// TwinCAT 3 PLC project PLC
// ProgramVersion: 3.1.4024.0
// libraries:
//   Tc2_Standard, * (Beckhoff Automation GmbH)
//   Tc2_System, * (Beckhoff Automation GmbH)
//   Tc3_Module, * (Beckhoff Automation GmbH)
// project tree:
//   / PlcTask1.TcTTO, PlcTask2.TcTTO
//   POUs/ MAIN_ST.TcPOU, MAIN_CFC.TcPOU, ProductionAnalytics.TcPOU
// real-time tasks:
//   TASK PlcTask1: cycle T#10ms, priority 20, ADS port 350
//   TASK PlcTask2: cycle T#10ms, priority 1, ADS port 351

CONFIGURATION PLC
    RESOURCE PLC ON TwinCAT3
        TASK PlcTask1(INTERVAL := T#10ms, PRIORITY := 20);
        TASK PlcTask2(INTERVAL := T#10ms, PRIORITY := 1);
        PROGRAM MAIN_ST WITH PlcTask1 : MAIN_ST;
        PROGRAM MAIN_CFC WITH PlcTask2 : MAIN_CFC;
    END_RESOURCE
END_CONFIGURATION

// ---- POUs/MAIN_ST.TcPOU
PROGRAM MAIN_ST
VAR
	ProductionAnalytics		:	ProductionAnalytics;
	UnsortArray		: ARRAY[1..10] OF REAL := [5, 3, 8, 5, 6, 5, 5, 23, 5, 9];
	SortedArray		: ARRAY[1..10] OF REAL;
	
	Sort			: BOOL;
	GetMean			: BOOL;
	GetStdDev		: BOOL;
	GetTotal		: BOOL;
	GetMax			: BOOL;
	GetMin			: BOOL;
	FindItem		: BOOL;
	Mean			: REAL;
	StdDev			: REAL;
	Total			: REAL;
	MaxItem			: REAL;
	MinItem			: REAL;
	FoundItemIdx	: UINT;
	ItemFound		: BOOL;
	ValidInput		: BOOL;
	IsSorted		: BOOL;
END_VAR

ProductionAnalytics(DataArray:=UnsortArray);
IF GetMean THEN
	Mean := ProductionAnalytics.GetMean();
ELSIF GetStdDev THEN
	StdDev := ProductionAnalytics.GetStdDev();
ELSIF GetTotal THEN
	Total := ProductionAnalytics.GetTotal();
ELSIF FindItem THEN
	ProductionAnalytics.FindItem( SearchValue := 23, StartIndex := 1, Endindex := 10,
								  FoundIndex => FoundItemIdx , 
								  Found => ItemFound, 
								  ValidInput => ValidInput);
ELSIF Sort THEN
	ProductionAnalytics.Sort(SortedArray => SortedArray, 
							 IsSorted => IsSorted, 
							 ValidInput => ValidInput);
ELSIF GetMax THEN
	MaxItem := ProductionAnalytics.GetMaxItem();

ELSIF GetMin THEN
	MinItem := ProductionAnalytics.GetMinItem();
END_IF

END_PROGRAM

// ---- POUs/ProductionAnalytics.TcPOU
FUNCTION_BLOCK ProductionAnalytics

VAR_IN_OUT
	DataArray 		: ARRAY[1..ARRAY_SIZE] OF REAL;   // Input array for analytics
END_VAR
VAR
	Idx       		: INT;                    		  // loop index 
END_VAR

VAR CONSTANT
	ARRAY_SIZE		: UINT := 10;
END_VAR

METHOD FindItem
VAR_INPUT
	SearchValue : REAL;             // The value to search for
    StartIndex  : UINT;            // Start index of the array to search in (1-based)
    EndIndex    : UINT;            // End index of the array to search in (1-based)
END_VAR

VAR_OUTPUT
    FoundIndex  : UINT;            // Index of the found value (1-based), 0 if not found
    Found       : BOOL;            // TRUE if the value is found, FALSE otherwise
    ValidInput  : BOOL;            // Indicates if the input parameters are valid
END_VAR

VAR
    MidIndex    : UINT;             // Midpoint index for binary search
    Low         : UINT;             // Lower boundary for search
    High        : UINT;             // Upper boundary for search
END_VAR
(* Find element using binary search algorithm *)

// Input validation
IF (StartIndex >= 1) AND (EndIndex <= ARRAY_SIZE) AND (StartIndex <= EndIndex) THEN
    ValidInput := TRUE;
ELSE
    ValidInput := FALSE;
    Found := FALSE;
    FoundIndex := 0;
    RETURN;
END_IF;

// Binary Search Algorithm
Low := StartIndex;
High := EndIndex;
Found := FALSE;       

WHILE (Low <= High) AND (NOT Found) DO
    // Calculate midpoint
    MidIndex := (Low + High) / 2;
    
    IF DataArray[MidIndex] = SearchValue THEN
        // Value found
        Found := TRUE;
        FoundIndex := MidIndex;
    ELSIF DataArray[MidIndex] < SearchValue THEN
        // Search in the right half
        Low := MidIndex + 1;
    ELSE
        // Search in the left half
        High := MidIndex - 1;
    END_IF;
END_WHILE;

// If not found, set FoundIndex to 0
IF NOT Found THEN
    FoundIndex := 0;  // Set to 0 to indicate not found
END_IF;
END_METHOD

METHOD GetMaxItem : REAL
VAR_INPUT
END_VAR

VAR
	ValidInput		: BOOL;
	SortedArray		: ARRAY[1..ARRAY_SIZE] OF REAL;
	IsSorted		: BOOL;
END_VAR
THIS^.Sort(SortedArray=>SortedArray, 
			IsSorted=>IsSorted, 
			ValidInput=>ValidInput);
			
If IsSorted then
	GetMaxItem := SortedArray[ARRAY_SIZE];
END_IF
END_METHOD

METHOD GetMean : REAL
VAR_INPUT
END_VAR

VAR
	Sum			: REAL;        // Sum of array elements 
	MeanTemp	: REAL;        // Temporary mean value for calculations
	Idx			: UINT;        // Loop counter 
END_VAR
(* Calculate the Mean *)

FOR Idx := 1 TO ARRAY_SIZE DO
	Sum := Sum + THIS^.DataArray[Idx];
END_FOR;


MeanTemp := Sum / TO_REAL(ARRAY_SIZE);
GetMean := MeanTemp;
END_METHOD

METHOD GetMinItem : REAL
VAR_INPUT
END_VAR

VAR
	ValidInput		: BOOL;
	SortedArray		: ARRAY[1..ARRAY_SIZE] OF REAL;
	IsSorted		: BOOL;
END_VAR
THIS^.Sort(SortedArray=>SortedArray, 
			IsSorted=>IsSorted, 
			ValidInput=>ValidInput);
			
If IsSorted then
	GetMinItem := SortedArray[1];
END_IF
END_METHOD

METHOD GetStdDev : REAL
VAR_INPUT
END_VAR

VAR
	MeanTemp		: REAL;		// Temporary mean value for calculations
	Deviation		: REAL;		// Deviation of each element from the mean
	SumOfSquares	: REAL;		// Sum of squared differences from the mean
	Idx				: UINT;     // Loop counter
	ArrayElement	: REAL;   	// Casted array element to REAL for precision
	MeanError		: BOOL;
END_VAR
(* Calculate the Standard Deviation *)

MeanTemp := THIS^.GetMean();

IF ARRAY_SIZE > 0 THEN
	FOR Idx := 1 TO ARRAY_SIZE DO
		ArrayElement := THIS^.DataArray[Idx];
		Deviation := ArrayElement - MeanTemp;						 
		SumOfSquares := SumOfSquares + (Deviation * Deviation); 
	END_FOR;

	GetStdDev := SQRT(SumOfSquares / TO_REAL(ARRAY_SIZE));
END_IF;
END_METHOD

METHOD GetTotal : REAL
VAR_INPUT
END_VAR

VAR
	Idx				: UINT;		// Loop counter
	ArrayElement	: REAL;		// Temporary array value	
	Total			: REAL;
END_VAR
FOR Idx := 1 TO ARRAY_SIZE DO
	ArrayElement := DataArray[Idx];
	Total := Total + ArrayElement;
END_FOR;

GetTotal := Total;
END_METHOD

METHOD Sort
VAR_INPUT
END_VAR

VAR_OUTPUT
    SortedArray   : ARRAY[1..ARRAY_SIZE] OF REAL;   // Output array with sorted elements
    IsSorted      : BOOL;                   // Indicates if the array is sorted
    ValidInput    : BOOL;                   // Indicates if the input parameters are valid
END_VAR

VAR
    Idx       	  : UINT;                   // Loop indices
    Parent, Child : UINT;                   // Indices for heap construction
    Temp          : REAL;                   // Temporary variable for swapping
END_VAR
(* Sort items using Heapsort algorithm*)

// --- Input Validation ---
IF (ARRAY_SIZE < 1) OR (ARRAY_SIZE > 100) THEN
    ValidInput := FALSE;
    IsSorted := FALSE;
    RETURN;
ELSE
    ValidInput := TRUE;
END_IF;

// --- Copy input array to output array ---
FOR Idx := 1 TO ARRAY_SIZE DO
    SortedArray[Idx] := THIS^.DataArray[Idx];
END_FOR;

// --- Heap Construction Phase ---
Idx := ARRAY_SIZE / 2;
WHILE Idx >= 1 DO
    Parent := Idx;
    WHILE 2 * Parent <= ARRAY_SIZE DO
        Child := 2 * Parent;
        
        // Select the larger child
        IF (Child < ARRAY_SIZE) AND 
			(SortedArray[Child] < SortedArray[Child + 1]) THEN
            Child := Child + 1;
        END_IF;
        
        // If parent is smaller than the largest child, swap them
        IF SortedArray[Parent] < SortedArray[Child] THEN
            Temp := SortedArray[Parent];
            SortedArray[Parent] := SortedArray[Child];
            SortedArray[Child] := Temp;
            
            // Move down the heap
            Parent := Child;
        ELSE
            EXIT;  // Break loop if the heap property is satisfied
        END_IF;
    END_WHILE;
    
    Idx := Idx - 1;  // Equivalent to DOWNTO without using DOWNTO
END_WHILE;

// --- Sorting Phase ---
FOR Idx := ARRAY_SIZE TO 2 BY -1 DO
    // Swap the first element (largest) with the last unsorted element
    Temp := SortedArray[1];
    SortedArray[1] := SortedArray[Idx];
    SortedArray[Idx] := Temp;
    
    // Restore the heap property for the reduced heap
    Parent := 1;
    WHILE 2 * Parent < Idx DO
        Child := 2 * Parent;
        
        // Select the larger child
        IF (Child < (Idx - 1)) AND (SortedArray[Child] < SortedArray[Child + 1]) THEN
            Child := Child + 1;
        END_IF;
        
        // If parent is smaller than the largest child, swap them
        IF SortedArray[Parent] < SortedArray[Child] THEN
            Temp := SortedArray[Parent];
            SortedArray[Parent] := SortedArray[Child];
            SortedArray[Child] := Temp;
            
            // Move down the heap
            Parent := Child;
        ELSE
            EXIT;  // Break loop if the heap property is satisfied
        END_IF;
    END_WHILE;
END_FOR;

// --- Set output signal to indicate sorting completion ---
IsSorted := TRUE;
END_METHOD

END_FUNCTION_BLOCK

// ---- POUs/MAIN_CFC.TcPOU
PROGRAM MAIN_CFC
VAR
	ProductionAnalytics		:	ProductionAnalytics;
	RawDataArray	: ARRAY[1..10] OF REAL := [5, 3, 8.3, 5, 6, 5, 5, 23, 5, 9];
	SortedArray		: ARRAY[1..10] OF REAL;
	
	Sort			: BOOL;
	GetMean			: BOOL;
	GetStdDev		: BOOL;
	GetTotal		: BOOL;
	GetMax			: BOOL;
	FindItem		: BOOL;
	Mean			: REAL;
	StdDev			: REAL;
	Total			: REAL;
	MaxItem			: REAL;
	FoundItemIdx	: UINT;
	ItemFound		: BOOL;
	ValidInput		: BOOL;
	IsSorted		: BOOL;
	ValueToFind		: REAL;
END_VAR

VAR CONSTANT
	ARRAY_SIZE		: UINT := 10;
END_VAR
VAR // added by the converter: edge detectors and wires of the graphical bodies
    _w1, _w2, _w3, _w4, _w5, _w6, _w7, _w8, _w9, _w10 : ANY;
END_VAR

ProductionAnalytics(DataArray := RawDataArray);
IF GetMean THEN _w1 := ProductionAnalytics.GetMean(); END_IF
Mean := _w1;
IF GetStdDev THEN _w2 := ProductionAnalytics.GetStdDev(); END_IF
StdDev := _w2;
IF GetTotal THEN _w3 := ProductionAnalytics.GetTotal(); END_IF
Total := _w3;
IF FindItem THEN ProductionAnalytics.FindItem(SearchValue := ValueToFind, StartIndex := 1, EndIndex := 10, FoundIndex => _w4, Found => _w5, ValidInput => _w6); END_IF
FoundItemIdx := _w4;
ItemFound := _w5;
ValidInput := _w6;
IF Sort THEN ProductionAnalytics.Sort(SortedArray => _w7, IsSorted => _w8, ValidInput => _w9); END_IF
SortedArray := _w7;
IsSorted := _w8;
ValidInput := _w9;
IF GetMax THEN _w10 := ProductionAnalytics.GetMaxItem(); END_IF
MaxItem := _w10;

END_PROGRAM
